KUKA KRL program: milling_2.src, milling_2.dat

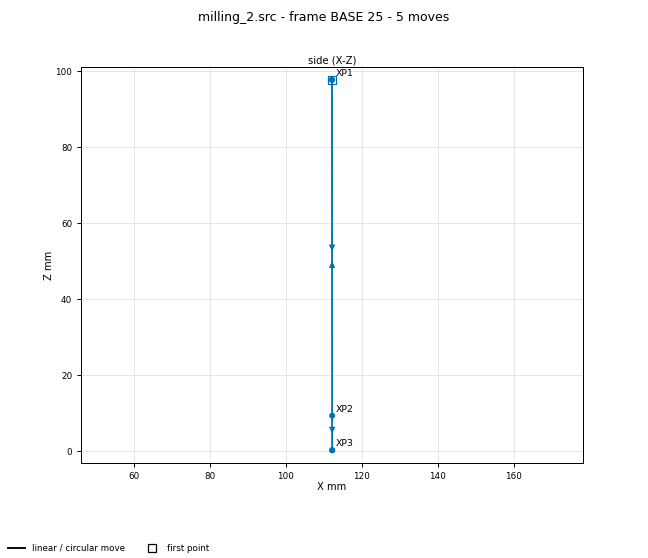
[picture p0: tool path of milling_2.src in frame BASE 25, 5 of 9 moves have a stored position in this frame; points joined in program order, loops and branches not executed]
--- milling_2.src ---
&ACCESS RVO
&REL 38
&PARAM EDITMASK = *
&PARAM TEMPLATE = C:\KRC\Roboter\Template\ExpertVorgabe
&PARAM DISKPATH = KRC:\R1\Program
DEF milling_2( )


SpindleRun(TRUE,9000,#CLOCKWISE)

wait sec 1
pos_d=xp3

;FOLD PTP P1 CONT Vel=30 % PDAT1 Tool[3]:Probe_Pin Base[25]:Base25;%{PE}
;FOLD Parameters ;%{h}
;Params IlfProvider=kukaroboter.basistech.inlineforms.movement.old; Kuka.IsGlobalPoint=False; Kuka.PointName=P1; Kuka.BlendingEnabled=True; Kuka.MoveDataPtpName=PDAT1; Kuka.VelocityPtp=30; Kuka.CurrentCDSetIndex=0; Kuka.MovementParameterFieldEnabled=True; IlfCommand=PTP
;ENDFOLD
$BWDSTART = FALSE
PDAT_ACT = PPDAT1
FDAT_ACT = FP1
BAS(#PTP_PARAMS, 30.0)
SET_CD_PARAMS (0)
PTP XP1 C_Dis
;ENDFOLD
;FOLD LIN P2 CONT Vel=0.1 m/s CPDAT1 Tool[3]:Probe_Pin Base[25]:Base25 ;%{PE}
;FOLD Parameters ;%{h}
;Params IlfProvider=kukaroboter.basistech.inlineforms.movement.old; Kuka.IsGlobalPoint=False; Kuka.PointName=P2; Kuka.BlendingEnabled=True; Kuka.MoveDataName=CPDAT1; Kuka.VelocityPath=0.1; Kuka.CurrentCDSetIndex=0; Kuka.MovementParameterFieldEnabled=True; IlfCommand=LIN
;ENDFOLD
$BWDSTART = FALSE
LDAT_ACT = LCPDAT1
FDAT_ACT = FP2
BAS(#CP_PARAMS, 0.1)
SET_CD_PARAMS (0)
LIN XP2 C_Dis C_Dis
;ENDFOLD
;FOLD LIN P3 CONT Vel=0.05 m/s CPDAT2 Tool[3]:Probe_Pin Base[25]:Base25 ;%{PE}
;FOLD Parameters ;%{h}
;Params IlfProvider=kukaroboter.basistech.inlineforms.movement.old; Kuka.IsGlobalPoint=False; Kuka.PointName=P3; Kuka.BlendingEnabled=True; Kuka.MoveDataName=CPDAT2; Kuka.VelocityPath=0.05; Kuka.CurrentCDSetIndex=0; Kuka.MovementParameterFieldEnabled=True; IlfCommand=LIN
;ENDFOLD
$BWDSTART = FALSE
LDAT_ACT = LCPDAT2
FDAT_ACT = FP3
BAS(#CP_PARAMS, 0.05)
SET_CD_PARAMS (0)
LIN XP3 C_Dis C_Dis
;ENDFOLD
$vel.cp=0.003
pos_d.z=pos_d.z-3.5
wait sec 0
$timer[1]=0
$timer_stop[1]=false
lin pos_d
;$base=base_data[25]
;$tool=tool_data[3]
x0_offset=pos_d.x
y0_offset=pos_d.y
z0_offset=pos_d.z
Rc=6


direc=true
if direc==true then
for ii=1 to 91
theta[ii]=(ii-1)*4.0
xy361[1,ii]=Rc*cos(theta[ii])+x0_offset
xy361[2,ii]=Rc*sin(theta[ii])+y0_offset
endfor
endif

cirp0.x=x0_offset
cirp0.y=y0_offset
cirp1.x=xy361[1,1]
cirp1.y=xy361[2,1]
$APO.CVEL=1
for ii=1 to 6
;$vel_axis[ii]=10
;$vel_axis[ii]=10
endfor
lin cirp1
kk=2
loop
cirp.x=xy361[1,kk]
cirp.y=xy361[2,kk]
lin cirp c_vel
kk=kk+1
if kk>=92 then

for ii=1 to 6
;$vel_axis[ii]=10
;$vel_axis[ii]=10
endfor
exit
endif
endloop

for ii=1 to 6
;$vel_axis[ii]=10
;$vel_axis[ii]=10
endfor





wait sec 0
$timer_stop[1]=true

$vel.cp=0.05
lin pos_d
lin xp3

;FOLD LIN P4 CONT Vel=0.3 m/s CPDAT3 Tool[3]:Probe_Pin Base[25]:Base25 ;%{PE}
;FOLD Parameters ;%{h}
;Params IlfProvider=kukaroboter.basistech.inlineforms.movement.old; Kuka.IsGlobalPoint=False; Kuka.PointName=P4; Kuka.BlendingEnabled=True; Kuka.MoveDataName=CPDAT3; Kuka.VelocityPath=0.3; Kuka.CurrentCDSetIndex=0; Kuka.MovementParameterFieldEnabled=True; IlfCommand=LIN
;ENDFOLD
$BWDSTART = FALSE
LDAT_ACT = LCPDAT3
FDAT_ACT = FP4
BAS(#CP_PARAMS, 0.3)
SET_CD_PARAMS (0)
LIN XP4 C_Dis C_Dis
;ENDFOLD
wait sec 1
SpindleRun(FALSE,0,#CLOCKWISE)
END

--- milling_2.dat ---
&ACCESS RVO
&REL 38
&PARAM EDITMASK = *
&PARAM TEMPLATE = C:\KRC\Roboter\Template\ExpertVorgabe
&PARAM DISKPATH = KRC:\R1\Program
DEFDAT  milling_2 PUBLIC


DECL E6POS pos_u,pos_d,cirp,cirp0,cirp1,cirp2,auxp1,auxp2
DECL BOOL direc
DECL REAL x0_offset,y0_offset,z0_offset,theta[91],xy361[2,361],xyz[3,6],Rc,A,B,Angle_x
DECL INT ii,jj,kk,Base_N
STRUC TUAN_TYP INT BASE_YUAN,REAL PHY



DECL E6POS XP1={X 112.131317,Y 16.1389217,Z 97.7742844,A 103.696251,B -0.733885407,C -1.60341465,S 22,T 51,E1 0.0,E2 0.0,E3 0.0,E4 0.0,E5 0.0,E6 0.0}
DECL FDAT FP1={TOOL_NO 3,BASE_NO 25,IPO_FRAME #BASE,POINT2[] " "}
DECL PDAT PPDAT1={VEL 30.0000,ACC 100.000,APO_DIST 500.000,APO_MODE #CDIS,GEAR_JERK 100.000,EXAX_IGN 0}
DECL MODULEPARAM_T LAST_TP_PARAMS={PARAMS[] "Kuka.PointName=P3; Kuka.FrameData.base_no=25; Kuka.FrameData.tool_no=3; Kuka.FrameData.ipo_frame=#BASE; Kuka.isglobalpoint=False; Kuka.MoveDataPtpName=PDAT1; Kuka.MovementDataPdat.apo_mode=#CDIS; Kuka.MovementDataPdat.apo_dist=500; Kuka.MovementData.vel=0.05; Kuka.MovementData.acc=100; Kuka.MovementData.exax_ign=0; Kuka.VelocityPtp=30; Kuka.BlendingEnabled=True; Kuka.APXEnabled=False; Kuka.CurrentCDSetIndex=0; Kuka.FrameData.point2=; Kuka.MoveDataName=CPDAT2; Kuka.MovementData.apo_fac=50; Kuka.MovementData.apo_dist=500; Kuka.MovementData.axis_acc=100; Kuka.MovementData.axis_vel=100; Kuka.MovementData.circ_typ=#BASE; Kuka.MovementData.jerk_fac=50; Kuka.MovementData.ori_typ=#VAR; Kuka.VelocityPath=0.05         "}
DECL E6POS XP2={X 112.182274,Y 16.1230221,Z 9.30554771,A 103.693611,B -0.735118270,C -1.60384107,S 22,T 51,E1 0.0,E2 0.0,E3 0.0,E4 0.0,E5 0.0,E6 0.0}
DECL FDAT FP2={TOOL_NO 3,BASE_NO 25,IPO_FRAME #BASE,POINT2[] " "}
DECL LDAT LCPDAT1={VEL 0.100000,ACC 100.000,APO_DIST 500.000,APO_FAC 50.0000,AXIS_VEL 100.000,AXIS_ACC 100.000,ORI_TYP #VAR,CIRC_TYP #BASE,JERK_FAC 50.0000,GEAR_JERK 100.000,EXAX_IGN 0}
DECL E6POS XP3={X 112.187668,Y 16.1221275,Z 0.217314929,A 103.693336,B -0.735254943,C -1.60389626,S 22,T 51,E1 0.0,E2 0.0,E3 0.0,E4 0.0,E5 0.0,E6 0.0}
DECL FDAT FP3={TOOL_NO 3,BASE_NO 25,IPO_FRAME #BASE,POINT2[] " "}
DECL LDAT LCPDAT2={VEL 0.0500000,ACC 100.000,APO_DIST 500.000,APO_FAC 50.0000,AXIS_VEL 100.000,AXIS_ACC 100.000,ORI_TYP #VAR,CIRC_TYP #BASE,JERK_FAC 50.0000,GEAR_JERK 100.000,EXAX_IGN 0}
DECL E6POS XP4={X 112.131317,Y 16.1389217,Z 97.7742844,A 103.696251,B -0.733885407,C -1.60341465,S 22,T 51,E1 0.0,E2 0.0,E3 0.0,E4 0.0,E5 0.0,E6 0.0}
DECL FDAT FP4={TOOL_NO 3,BASE_NO 25,IPO_FRAME #BASE,POINT2[] " "}
DECL LDAT LCPDAT3={VEL 0.300000,ACC 100.000,APO_DIST 500.000,APO_FAC 50.0000,AXIS_VEL 100.000,AXIS_ACC 100.000,ORI_TYP #VAR,CIRC_TYP #BASE,JERK_FAC 50.0000,GEAR_JERK 100.000,EXAX_IGN 0}
ENDDAT
